{attribute 'linkalways'} 
{attribute 'no_explicit_call' := 'This FB is a CLASS and must be accessed using methods or properties'}
{attribute 'enable_dynamic_creation'}
FUNCTION_BLOCK _ETcVnKeypointDetectionTypeFAST EXTENDS EnumDatatypeBase
VAR
	localData : ETcVnKeypointDetectionTypeFAST;
	activeData : REFERENCE TO ETcVnKeypointDetectionTypeFAST;
	enumBaseDatatype : _DINT(localData);
END_VAR

METHOD PRIVATE AddLocalEnumeration
VAR_INPUT
	Enumeration : T_MAXSTRING;
	Value : ETcVnKeypointDetectionTypeFAST;
END_VAR
AddEnumeration(Enumeration, Value);
END_METHOD

PROPERTY PUBLIC Address : PVOID
GET
Address := ADR(activeData);
END_GET
END_PROPERTY

METHOD PUBLIC ClearReference
VAR_INPUT
END_VAR
activeData REF= localData;
SetBaseDatatypeReference();
END_METHOD

METHOD PUBLIC Clone : I_Datatype
VAR
    pClone : POINTER TO _ETcVnKeypointDetectionTypeFAST;
END_VAR
pClone := __NEW(_ETcVnKeypointDetectionTypeFAST(InitialValue := Value));
Clone := pClone^;
END_METHOD

METHOD FB_init : BOOL
VAR_INPUT
	bInitRetains : BOOL; // if TRUE, the retain variables are initialized (warm start / cold start)
	bInCopyCode : BOOL;  // if TRUE, the instance afterwards gets moved into the copy code (online change)
	InitialValue : ETcVnKeypointDetectionTypeFAST;
END_VAR
localData := InitialValue;
AddBaseDatatype(enumBaseDatatype);
ClearReference();

AddLocalEnumeration('TCVN_KDT_FAST_5_8', ETcVnKeypointDetectionTypeFAST.TCVN_KDT_FAST_5_8);
AddLocalEnumeration('TCVN_KDT_FAST_7_12', ETcVnKeypointDetectionTypeFAST.TCVN_KDT_FAST_7_12);
AddLocalEnumeration('TCVN_KDT_FAST_9_16', ETcVnKeypointDetectionTypeFAST.TCVN_KDT_FAST_9_16);
END_METHOD

PROPERTY PUBLIC Identifier : T_MAXSTRING
GET
Identifier := 'ETcVnKeypointDetectionTypeFAST';
END_GET
END_PROPERTY

METHOD IsEnumeratorValueEqual : BOOL
VAR_INPUT
	Enumerator : I_KeyValueForwardEnumerator;
END_VAR
VAR
	storedValue : ETcVnKeypointDetectionTypeFAST;
END_VAR
IF NOT Enumerator.TryGet(storedValue) THEN
	RETURN;
END_IF

IsEnumeratorValueEqual := storedValue = activeData;
END_METHOD

METHOD PUBLIC MakeReferenceTo
VAR_INPUT
	ReferenceTarget : REFERENCE TO ETcVnKeypointDetectionTypeFAST;
END_VAR
activeData REF= ReferenceTarget;
SetBaseDatatypeReference();
END_METHOD

METHOD PROTECTED SetBaseDatatypeReference
VAR_INPUT
END_VAR
enumBaseDatatype.MakeReferenceTo(activeData);
END_METHOD

PROPERTY PUBLIC Size : UDINT
GET
Size := SIZEOF(activeData);
END_GET
END_PROPERTY

METHOD TryMakeReferenceTo : BOOL
VAR_INPUT
	Target : I_Datatype;
END_VAR
VAR
	targetAsEnum : I_EnumDatatype;
	pTargetData : POINTER TO ETcVnKeypointDetectionTypeFAST;
END_VAR
IF NOT Target.TryResolveAsEnumDatatype(targetAsEnum) THEN
	RETURN;
END_IF

IF targetAsEnum.Identifier <> Identifier THEN
	RETURN;
END_IF

pTargetData := Target.Address;
activeData REF= pTargetData^;
SetBaseDatatypeReference();
TryMakeReferenceTo := TRUE;
END_METHOD

PROPERTY PUBLIC Value : ETcVnKeypointDetectionTypeFAST
GET
Value := activeData;
END_GET
SET
activeData := Value;
END_SET
END_PROPERTY

END_FUNCTION_BLOCK

(* stored: Version 1.1.0.1, ProductVersion 3.1.4024.13
   POU _ETcVnKeypointDetectionTypeFAST: Id {9db57aa0-3898-0c5e-0a3b-868c16e81042}, SpecialFunc None
   Folder Core: Id {15954782-1a09-02e8-02a9-cb59f3ffd44e}
   Folder Protected: Id {fe3a3bc4-0046-0a65-2165-8d796685aebd}
   Folder Customize: Id {cf71291e-b1d0-015f-2a8a-613005a7217d}
   Folder Constructor: Id {292e28be-2a1b-0d12-1aeb-5927446aa30e}
   Folder Private: Id {16698e31-6beb-0d1e-085a-251c5be8ee87}
   Folder Protected: Id {cf08ea19-73ca-0d53-0f90-73da85da43b4}
   Method AddLocalEnumeration: Id {bae865cd-0ca8-052f-2e3e-b5c76d81c1f3}
   Property Address: Id {3a4eaca8-f942-036a-344f-4a2ec7460972}
   Get Get: Id {f587e5c0-214a-05aa-2aac-6eaee4760faa}
   Method ClearReference: Id {8b46238b-8972-06c3-226b-036d2a9284a8}
   Method Clone: Id {d404555d-b0c9-0cee-1a81-15addfc394b2}
   Method FB_init: Id {1f280970-f67d-023f-2cd3-20f72caa8b6f}
   Property Identifier: Id {d49ea7e0-5acc-0928-0ed1-4a11aa55f4de}
   Get Get: Id {37828915-15ca-0ba7-09c0-7d2a9afcf09a}
   Method IsEnumeratorValueEqual: Id {d2140e97-7a78-0d8f-3cc7-1ca4d348746a}
   Method MakeReferenceTo: Id {34358bb1-6fa8-05df-0982-5a7f8d1522be}
   Method SetBaseDatatypeReference: Id {316d8493-dc5d-077a-22b9-92ccb31fa565}
   Property Size: Id {55a66f05-2ee0-0063-278b-95349dc91b27}
   Get Get: Id {2dc75ecd-d26c-0e50-2385-54a09dada034}
   Method TryMakeReferenceTo: Id {a2f1488f-02f5-0c5f-18da-872677387083}
   Property Value: Id {86635275-8d5e-088b-20a3-02be4a154ca2}
   Get Get: Id {aec4a33e-8846-0345-2908-49b4b5fcd258}
   Set Set: Id {a64d5ed6-0337-0655-11a6-4c9d54847f1d} *)
